PROGRAM Planar_Mover
VAR
	
fbMover 					:		ARRAY [1..2]  OF MC_PlanarMover ; // Change based on how many movers there are
cmdFB 						:		ARRAY [1..2]  OF MC_PlanarFeedBack ; 
stMoverPositions 			:		ARRAY [1..12] OF PositionXYC ;
fbDynMove					:		ARRAY [1..5]  OF DynamicConstraint_PathXY ;
stExtOptions				:		ARRAY [1..2]  OF ST_ExternalSetpointGenerationOptions; 
Done						: 	 	BOOL;
nCase						: 		INT := 1;
timer						: 		TON;
moverState					:		MC_Planar_State; 
RESET						: 		BOOL;


END_VAR

//Mover 1 updates
fbMover[1].Update(); 
cmdFB[1].Update();
moverState := fbMover[1].MCTOPLC.STD.State;

Timer(IN := TRUE, PT := T#1S); 

IF Timer.Q THEN
	//Start initizalization
	IF NOT done OR MoverState = 5 OR MoverState = 1 THEN 
		Planar_Mover.init();
	END_IF 
END_IF

METHOD init 
VAR_INPUT
END_VAR

VAR


END_VAR
CASE nCase OF
1: 
	//fbmover[1].StopExternalSetpointGeneration(cmdFb[1]);
	Done := FALSE;
	fbMover[1].Reset(cmdFB[1]);
	//fbMover[2].Reset(cmdFB[2]);
	nCase := 2;

2:

	IF cmdFB[1].Done THEN
		nCase := 3; 
	END_IF
	
3:

	fbMover[1].Enable(cmdFB[1]);
	nCase := 4;
	
4:

	IF cmdFB[1].Done THEN
		nCase := 5;
	END_IF
	
5:

//Set up Case
	// Setting Movingg Positions 
	stMoverPositions[5].SetValuesXYC(120,360,0); // Mover 1 Start 

	// Normal Movememnt
	fbDynMove[1].SetValuesVADJ(500,5000,5000,20000); // Normal
	fbDynMove[2].SetValuesVADJ(1000,5000,5000,20000);// Fast
	fbDynMove[3].SetValuesVADJ(200,2000,5000,10000); // Slow

	stExtOptions[1].mode := MC_EXTERNAL_SET_POSITION_MODE.Absolute; // Setting up external Setpoint generator
	nCase := 6; 
6:

Done := TRUE; 
nCase := 7;

7:

IF MoverState = 5 OR MoverState = 1 THEN
	IF XboxController.XboxController1.P_Buttons.bBack OR RESET THEN
		Constraints.Restarting := TRUE;  
		nCase := 1;	
	END_IF
END_IF 

	
END_CASE
END_METHOD

END_PROGRAM

(* stored: Version 1.1.0.1, ProductVersion 3.1.4024.12
   POU Planar_Mover: Id {aae6372a-0f1a-4d4a-a894-f979094bfc48}, SpecialFunc None
   Method init: Id {a476209f-a9e9-4db8-8329-893240eac645} *)
